TYPE U_OdriveEncoderEstimatesBytes :
UNION
    stEncoderEstimates : ST_OdriveEncoderEstimates;
    aBytes : ARRAY[0..7] OF BYTE;
END_UNION
END_TYPE

(* stored: Version 1.1.0.1
   DUT U_OdriveEncoderEstimatesBytes: Id {3da78d05-d5c7-46ef-a1a1-58725a104d68} *)
